INTERFACE I_HE_SATT_FilterHolderSelector


METHOD CoupleHolders
VAR_INPUT
    abCoupledHolders : ARRAY[1..PL_HE_SATT_Parameters.nNumHolders] OF BOOL;
END_VAR
END_METHOD


METHOD CouplingRulesSatisfied : BOOL
VAR_INPUT
    iFilterCombination : I_HE_SATT_FilterCombination;
END_VAR
END_METHOD


METHOD DeselectHolder
VAR_INPUT
    nHolderNumber : INT;
END_VAR
END_METHOD


METHOD IsSelected : BOOL
VAR_INPUT
    nHolderNumber : INT;
END_VAR
END_METHOD


METHOD Reset
END_METHOD


METHOD SelectHolder
VAR_INPUT
    nHolderNumber : INT;
END_VAR
END_METHOD

END_INTERFACE

(* stored: Version 1.1.0.1
   Itf I_HE_SATT_FilterHolderSelector: Id {2309a12e-dd09-4cf7-84a3-3982b60eb98c}
   Method CoupleHolders: Id {eaf3069d-83bc-4894-ad0f-850f60b111b0}
   Method CouplingRulesSatisfied: Id {c342b068-1c89-42b6-920f-2e9b123699f7}
   Method DeselectHolder: Id {31578d46-5b1a-451b-9ce8-c7bd877a8e4a}
   Method IsSelected: Id {dfc29f85-3adb-491a-90a0-3fea9c02e137}
   Method Reset: Id {211a3934-fc1b-4d02-8536-5d9a93e4035d}
   Method SelectHolder: Id {269cef13-4783-4c78-b9a9-5596ef9fb147} *)
